// Implicitly generated code : DO NOT EDIT
FUNCTION CheckDivReal : REAL
VAR_INPUT
	divisor:REAL;
END_VAR

// Implicitly generated code : Only an Implementation suggestion
{noflow}
IF divisor = 0 THEN
GVL_Checks.diCheckDivReal := GVL_Checks.diCheckDivReal +1;
	CheckDivReal:=1;
ELSE
	CheckDivReal:=divisor;
END_IF;
{flow}

END_FUNCTION

(* stored: Version 1.1.0.1, ProductVersion 3.1.4024.12
   POU CheckDivReal: Id {a98b279b-b1ed-454e-82d7-358ac55c00d5}, SpecialFunc CheckDivReal32 *)
